FUNCTION_BLOCK RejectMsgHandling
VAR_INPUT
	bReject			: BOOL;
	bRejectID		: INT;
	RejectType		: STRING;
	Counter			: UINT;
	RejectMsg		: STRING;
	Timestamp		: STRING;	
	bResetBuffer	: BOOL;
END_VAR
VAR_OUTPUT
END_VAR
VAR_IN_OUT
	dtRejectHistory	: ARRAY [1..20] OF stRejectData;
END_VAR
VAR
	i				: UINT;
	j				: UINT;
	LastIndex		: UINT;
	EmptyArray		: ARRAY [1..20] OF stRejectData;
	SeqIndex		: UINT;
	
END_VAR


	CASE SeqIndex OF
		0:
			IF bReject THEN
				SeqIndex	:= 5;	
			END_IF
			
		5:
			FOR i := 1 TO 20 BY 1 DO
			IF dtRejectHistory[i].Status = 0 THEN
				LastIndex	:= i;
				SeqIndex	:= 10;
				EXIT;
			END_IF
			END_FOR
				
			IF i > 20 THEN
				SeqIndex	:= 10;
			END_IF
			
			
		10:
			IF LastIndex > 1 THEN
				FOR j := LastIndex TO 2 BY -1 DO
					dtRejectHistory[j].Status		:=	dtRejectHistory[j-1].Status;
					dtRejectHistory[j].RejectID		:=	dtRejectHistory[j-1].RejectID;
					dtRejectHistory[j].RejectType	:=	dtRejectHistory[j-1].RejectType;
					dtRejectHistory[j].Counter		:=	dtRejectHistory[j-1].Counter;
					dtRejectHistory[j].RejectMsg	:=	dtRejectHistory[j-1].RejectMsg;
					dtRejectHistory[j].Timestamp	:=	dtRejectHistory[j-1].Timestamp;
				END_FOR
			END_IF
			
			//IF j >= LastIndex THEN
				SeqIndex	:= 20;
			//END_IF
			
		20:
				dtRejectHistory[1].Status			:=	1;
				dtRejectHistory[1].RejectID			:=	bRejectID;
				dtRejectHistory[1].RejectType		:=	RejectType;
				dtRejectHistory[1].Counter			:=	Counter+1;
				dtRejectHistory[1].RejectMsg		:=	RejectMsg;
				dtRejectHistory[1].Timestamp		:=	Timestamp;
				IF NOT bReject THEN
					i			:= 0;
					j			:= 0;
					SeqIndex	:= 0;
				END_IF
			
	END_CASE
	

IF bResetBuffer	THEN //OR LastIndex >= 20
	LastIndex		:= 0;
	i				:= 0;
	j				:= 0;
	SeqIndex		:= 0;
	dtRejectHistory	:= EmptyArray;
END_IF

END_FUNCTION_BLOCK

(* stored: Version 1.1.0.1, ProductVersion 3.1.4024.12
   POU RejectMsgHandling: Id {f9eb4f63-f2c6-4b6e-bf8e-ae2cf46d26c9}, SpecialFunc None *)
